Fanuc KAREL source: kb00149.KL

-- PROVISIONAL review KL for V1013-1; original PC SHA256 d8df303a5b5d485e83c530f5c52abee96b99d52751653791cd2f0db30fb64195
-- Incomplete behavior may be omitted. Consult companion uncertainty JSON. Do not deploy.
PROGRAM KB00149
%NOLOCKGROUP
BEGIN
  -- UNRESOLVED_PC offsets 5-12; opcodes 9D,23
  -- UNRESOLVED_PC offsets 17-27; opcodes 27,22,31
  -- UNRESOLVED_PC offsets 32-36; opcodes 7F
END KB00149
